// This function has been automatically generated from the project information.
{attribute 'signature_flag' := '1073741824'}
{attribute 'TcGenerated'}
{attribute 'no-analysis'}
FUNCTION F_GetCompany : WSTRING
VAR_INPUT
	
END_VAR

F_GetCompany := "Timberline Automation and Control Co.";

END_FUNCTION

(* stored: Version 1.1.0.1, ProductVersion 3.1.4026.12
   POU F_GetCompany: Id {ea05b85d-a6d5-4f46-87e2-f9c313de8eb7}, SpecialFunc None *)
